// TIA Portal V18 export
DATA_BLOCK "defects_util_DB"   // DB37
VERSION : 0.1
// stored: AutoNumber true, DBAccessibleFromOPCUA true, InstanceOfName defects_util, InstanceOfType FB
"defects_util"
   // VAR_INPUT
   //    ALLOWED : Bool;
   //    xBdefect_inc : Bool;
   //    xBdefect_dec : Bool;
   //    xDefectsClearAll : Bool;
   //    xDefect_Save : Bool;
   //    positions : "typePositions";
   // END_VAR
   // VAR_OUTPUT
   //    go_to_defect_now : Bool;
   // END_VAR
   // VAR_IN_OUT
   //    xyBeepDone : Bool;
   //    DEFECTS_DB : "typeDefectsDB";
   // END_VAR
   // VAR
   //    mem1 : Bool;
   //    mem2 : Bool;
   //    xdefect_dec_was : Bool;
   //    xdefect_inc_was : Bool;
   //    xDefect_Save_was : Bool;
   //    xDefectsClearAll_was : Bool;
   // END_VAR
BEGIN
END_DATA_BLOCK
